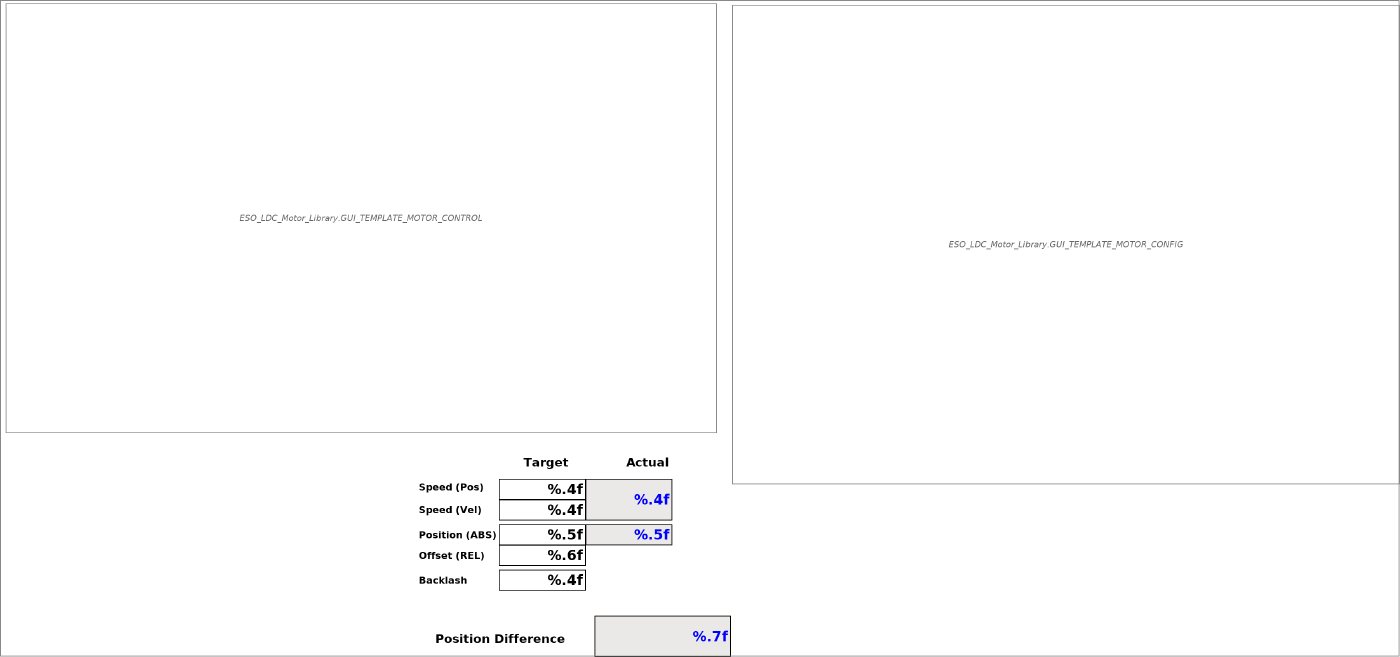
VISUALIZATION GUI_DL_2  // 1698x797
    Frame (7,4 862x521)
        shows ESO_LDC_Motor_Library.GUI_TEMPLATE_MOTOR_CONTROL(m_Instance := MAIN.DL_2)
    Frame (888,6 810x581)
        shows ESO_LDC_Motor_Library.GUI_TEMPLATE_MOTOR_CONFIG(m_Instance := MAIN.DL_2)
    Rectangle (505,581 95x20), "Speed (Pos)"
    Rectangle (710,636 105x25), "%.5f", text variable: MAIN.DL_2.stat.lrPosActual, input disabled if: false
    Rectangle (632,551 190x20), "Target Actual"
    Rectangle (505,639 95x20), "Position (ABS)"
    Rectangle (710,581 105x50), "%.4f", text variable: MAIN.DL_2.stat.lrVelActual, input disabled if: false
    Rectangle (605,606 105x25), "%.4f", text variable: MAIN.DL_2.ctrl.lrVelocity
        OnMouseDown: write the text variable via Default
    Rectangle (505,694 95x20), "Backlash"
    Rectangle (605,691 105x25), "%.4f", text variable: MAIN.DL_2.cfg.lrBacklash
        OnMouseDown: write the text variable via Default
    Rectangle (505,606 95x25), "Speed (Vel)"
    Rectangle (605,636 105x25), "%.5f", tooltip "Absolute position used by "MOVE ABS"", text variable: MAIN.DL_2.ctrl.lrPosition
        OnMouseDown: write the text variable via Default
    Rectangle (605,581 105x25), "%.4f", text variable: MAIN.DL_2.cfg.lrDefaultVelocity
        OnMouseDown: write the text variable via Default
    Rectangle (505,664 95x20), "Offset (REL)"
    Rectangle (605,661 105x25), "%.6f", tooltip "Relative offset used by "MOVE REL"", text variable: MAIN.DL_2.ctrl.lrOffset
        OnMouseDown: write the text variable via Default
    Rectangle (721,747 165x50), "%.7f", text variable: MAIN.DL_2.stat.lrPosError, input disabled if: false
    Rectangle (525,765 190x20), "Position Difference"
END_VISUALIZATION

(* stored: Version 1.1.0.1, ProductVersion 3.1.4024.12
   Visu GUI_DL_2: Id {0db1472b-0fd5-41dc-83d8-50204657af54} *)
